{attribute 'GeneratedUsingTerminal: EP9128-0021-0017'}
{attribute addProperty BoxType "EP9128-0021-0017"}
{attribute addProperty Id "A_0010_EP9128_0021_0018A_0010_EP9128_0021_0018_8540EC37527A_0007_EP9128_0021_0017_2_EP9128_1021EP9128_1FC0878B2A_0007_EP9128_0021_0017_3_EP9128_2021EP9128_1FC0878B2"}
{attribute addProperty CRC "2934543232"}
{attribute addProperty Size "531"}
TYPE A_0007_EP9128_0021_0017_AEE99380 EXTENDS EP9128_1FC0878B :
STRUCT
	{attribute addProperty Name "A_0010_EP9128_0021_0018"}
	{attribute addProperty PreviousPort "A_0007(EP9128-0021-0017) : D"}
	A_0010_EP9128_0021_0018 : A_0010_EP9128_0021_0018_8540EC37;
	{attribute addProperty Name "A_0007_EP9128_0021_0017_2_EP9128_1021"}
	{attribute addProperty PreviousPort "A_0007(EP9128-0021-0017) : C"}
	A_0007_EP9128_0021_0017_2_EP9128_1021 : EP9128_1FC0878B;
	{attribute addProperty Name "A_0007_EP9128_0021_0017_3_EP9128_2021"}
	{attribute addProperty PreviousPort "A_0007(EP9128-0021-0017)_2 (EP9128-1021) : C"}
	A_0007_EP9128_0021_0017_3_EP9128_2021 : EP9128_1FC0878B;
END_STRUCT
END_TYPE

(* stored: Version 1.2.0.0, ProductVersion 3.1.4024.9
   DUT A_0007_EP9128_0021_0017_AEE99380: Id {f043b517-d10b-48f6-9fbb-26bb7101b256} *)
